Fanuc KAREL source: kt00638.KL

-- PROVISIONAL review KL for V1013-1; original PC SHA256 7efa6aeb4e35c0177aaeb4559045db1d94bd2808d1b90896e5579f6d6df44961
-- Incomplete behavior may be omitted. Consult companion uncertainty JSON. Do not deploy.
PROGRAM KT00638
%NOLOCKGROUP
VAR
  OUT : REAL
-- UNRESOLVED_DECL Y1 type=002018
-- UNRESOLVED_DECL Y2 type=002018
BEGIN
  -- UNRESOLVED_PC offsets 5-19; opcodes 2E,22,9D,33,B2
  -- UNRESOLVED_PC offsets 24-38; opcodes 2E,22,9D,33,B2
  -- UNRESOLVED_PC offsets 43-57; opcodes 2E,22,9D,33,B2
  -- UNRESOLVED_PC offsets 62-76; opcodes 2E,22,9D,33,B2
  -- UNRESOLVED_PC offsets 81-97; opcodes 22,9D,33,B1,64,23
  -- UNRESOLVED_PC offsets 102-106; opcodes 7F
END KT00638
